{attribute 'GeneratedUsingTerminal: EL3443-0000-0017'}
{attribute addProperty BoxType "EL3443-0000-0017"}
{attribute addProperty Id "L1_L2_VoltageAT %I*REAL4L2_L3_VoltageAT %I*REAL4L3_L1_VoltageAT %I*REAL4"}
{attribute addProperty CRC "679556377"}
{attribute addProperty Size "12"}
TYPE Total_Total_L_L_Voltage_28813519 EXTENDS InputBase_8311D824 :
STRUCT
	{attribute addProperty Name "L1_L2_Voltage"}
	L1_L2_Voltage AT %I* : REAL;
	{attribute addProperty Name "L2_L3_Voltage"}
	L2_L3_Voltage AT %I* : REAL;
	{attribute addProperty Name "L3_L1_Voltage"}
	L3_L1_Voltage AT %I* : REAL;
END_STRUCT
END_TYPE

(* stored: Version 1.2.0.0, ProductVersion 3.1.4024.11
   DUT Total_Total_L_L_Voltage_28813519: Id {e0083d93-eac6-4461-a5db-414ee6182794} *)
